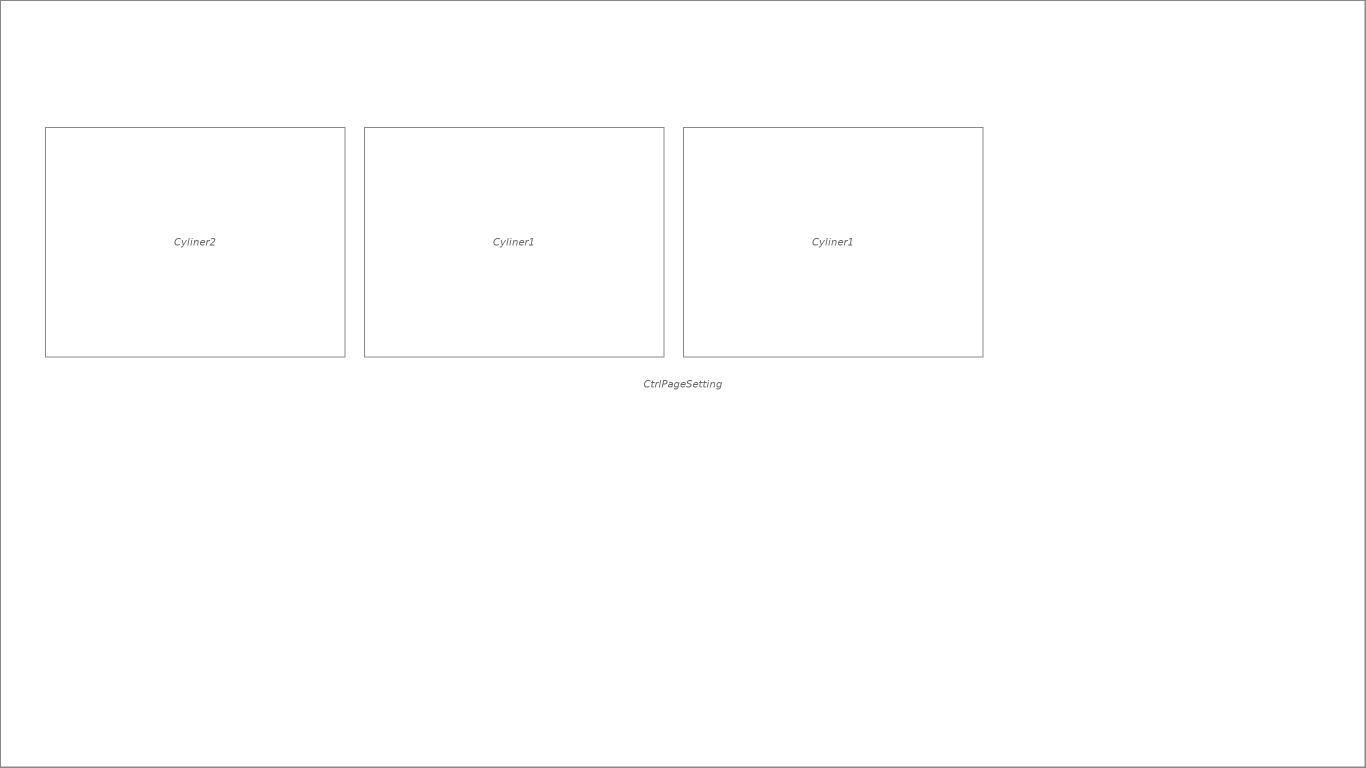
VISUALIZATION PageSetting_UnloadFrock  // 1366x768
    Frame (0,0 1366x768)
        shows CtrlPageSetting()
    Frame (683,127 300x230)
        shows Cyliner1(System := G_stSystem, Cylinder := G_arrCylinder[E_Cylinder.UnloadFrockLift], CylinderData := G_arrCylinderData[E_Cylinder.UnloadFrockLift])
    Frame (364,127 300x230)
        shows Cyliner1(System := G_stSystem, Cylinder := G_arrCylinder[E_Cylinder.UnloadFrockPrevent], CylinderData := G_arrCylinderData[E_Cylinder.UnloadFrockPrevent])
    Frame (45,127 300x230)
        shows Cyliner2(System := G_stSystem, Cylinder := G_arrCylinder[E_Cylinder.UnloadFrockPush], CylinderData := G_arrCylinderData[E_Cylinder.UnloadFrockPush])
END_VISUALIZATION

(* stored: Version 1.1.0.1, ProductVersion 3.1.4024.3
   Visu PageSetting_UnloadFrock: Id {a3e1cb77-4467-4854-84d5-092142526a2f} *)
